(*
Nazwa:			FB_CapFeederV2
Opis:			Sorter nasadek i podajnik nasadek z podnośnikiem JIESANG
Wersja:			v0.1
Data:			2022-07-07
Autor:			DJA
Urzadzenia:		Silnik sortera, podnośnik JIESANG, Wydmuch, czujniki zapełnienia rękawa
Konfiguracja:	
Info:
-poprawiona wersja sortera względem poprzedniej, przerobione na aktualny standard State i RunningState
*)


FUNCTION_BLOCK FB_CapFeeder_old
VAR_INPUT
	
	bEnable						: BOOL;					//Zezowlenie na pracę stacji sprawdzania
	bEStop						: BOOL;					//Stop Awaryjny nieaktywny
	bRun						: BOOL;					//Włączenie sortera nasadek
	bHoming						: BOOL;					//Zezwolenie na wykonanie bazowania i pozycjonowania stacji sprawdzania
	bHeightSet					: BOOL;					// Bit do bazowania stacji na ustaloną wysokość 
	bIgnoreError				: BOOL;					//Ignorowania błędów cyklu pracy
	bReset						: BOOL;					//Reset błędu, jeśli w stanie "eError"
	lrHeightMotorPositionSV		: LREAL;				//Wysokość zadana na której ma znajdować się stacja
	lrMaxHeight					: LREAL;				//Maksymalna wysokość stacji sprawdzania
	lrMinHeight					: LREAL;				//Minimalna wysokość stacji sprawdzania
	bSorterCapSensor 			: BOOL;					// Wejście z czujnika ultradzwiękowego nasadki sortera
	bFullSleeveSensor			: BOOL;					// Wejście przepełnienia rękawa sortera
	bLevelSensor				: BOOL;					// Czujnik poziomu
	bHomingSensor				: BOOL;					// Wejscie czujnika bazowania napedu 
	iTimeDelayOn				: INT; 					//Czas na właczenie silnika sortera po zaniku sygnału przepełnienia z rękawa
	iTimeDelayOff				: INT; 					// Czas na wylączenie silnika sortera po wykryciu sygnału przepełnienia z rękawa sortera
	iTimeToEmptySleeveError		: INT;					// Czas do włączenia alrmu pustego rękawa
	bEngineOK					: BOOL;					//Wejście czujnika zabezpieczenia silnika 
	InEngineVelocityCV 			: UDINT;		
	InEngineSTW 				: UINT; 				// Statusword transportera wejściowo wyjściowego
	IbEngineWcState				: BOOL; 				// Statusword transportera wejściowo wyjściowego
	bHeightMotorEncoderPulse 	: BOOL;					//Sygnał impulsów enkodera siłownika
	rHeightMotorPositionOffset 	: REAL;					//Wysokość bazowania podnośnika
	bManualMovement				: BOOL; 				//Uruchomienie trybu ruchów ręcznych
	udiStationIndex				: UDINT;				// Indywidualny numer stacji
	sStationName				: STRING;				// Nazwa stacji
	
	tGatesFreq					:	TIME;
	
	bSensorInPipe				:	BOOL;				// Czujnik obecnośći flipflopa w rękawie
END_VAR

VAR_OUTPUT
	eState						: E_Station;			// Aktualny stan stacju
	eRunningState				: E_CapFeederState;		// Stan pracy stacji
	eRunningStateBeforeEstop	: E_CapFeederState;  	// Stan przed Estope
	bError						: BOOL;					// Błąd stacji
	udiErrorID					: UDINT;				// Nr blędu przeciągania formatek
	sErrorDescription			: STRING(200);			// Opis błędu
	sErrorDescription2			: STRING(200);			// Opis błędu
	sErrorStationName			: STRING;				// Nazwa stacj
	udiStationID				: UDINT;				// Nr stacji

	lrHeightMotorPositionCV		: LREAL;				//Aktualna pozycja podnośnika stacji
	bHeightMotorUp				: BOOL;					//Sterowanie silnikiem podnośnika  - RUCH W GÓRĘ
	bHeightMotorDown			: BOOL;					//Sterowanie silnikiem podnośnika  - RUCH W DÓŁ
	bSorterEngine 				: BOOL; 				// Sterowanie silnikiem sortera
	QnEngineVelocitySV 			: UDINT; 				// Nastawa prędkości
	QnEngineCTW 				: UINT;  				// Controlword transportera we/wy	
	bSorterAir 					: BOOL; 				// Sterowanie szybkim zaworem wydmuchu
	bHomingNeeded				: BOOL;					// Wymagane ponowne bazowanie (blad podczas bazowania lub stop awaryjny)
	bHomingDone					: BOOL;					// Stacja zbazowana 
	bCycleDone					: BOOL;					// Sygnał o zakończeniu cyklu
	bCycleNotDone				: BOOL;					// Sygnał o niezakończonym cyklu
	tCycleTime					: TIME;	 				// Czas cyklu 
	sWarningDescription			: STRING;
	bWarning1					: BOOL;
	udiWarningID				: UDINT;
	
	bGate1						:	BOOL;	//Szlaban w podajniku nakrętek #1
	bGate2						:	BOOL;	//Szlaban w podajniku nakrętek #2
	
END_VAR

VAR_IN_OUT
	bManualHeightMotorUp		: BOOL;					//Ruch ręczny podnośnika stacji w górę
	bManualHeightMotorDown		: BOOL;					//Ruch ręczny podnośnika stacji w dół
	bManualSorterEngine			: BOOL;					//Ręczne włączenie silnika sortera
	bManualSorterAir			: BOOL;					//Ręczne włączenie zaworu wydmuchu
	
	bManualGate1				:	BOOL;									// Szlaban #1 w rękawe
	bManualGate2				:	BOOL;									// Szlaban #2 w rękawe		
END_VAR

VAR
	i							:	INT;
	aBufferedSensorValue		:	ARRAY[0..50] OF BOOL;	
	iValvesCycleCase			:	INT;
	rtOutSensor					:	R_TRIG;

	// State
	eLastState					: E_Station;			//Stan ogólny bloku
	eLastStateTemp				: E_Station;			//Stan ogólny bloku
	eLastRunningState			: E_CapFeederState;		//Stan podbloku
	eLastRunningStateTemp		: E_CapFeederState;		//Stan podbloku

	fbHeightMotorEncoder		: FB_JiesangActuatorEncoder;				// Blok enkodera podnośnika chwytaka stabilizującego pod zakręcarką	
	bHeightMotorEncoderCounterReset						:BOOL; 				// Sygnał resetu enkodera
	lrLastHeightMotorPositionCV		: LREAL;				// Pozycja podnośnika w poprzednim cyklu programu
	bHeightMotorEncoderHomed	: BOOL;					// Informacja od enkodera że jest zbazowany		
	bStateError					: BOOL;
	
	tofHeightMotorDown			: TOF;					// Opóźnienie ruchu w dół, żeby nie przeciązać rozruchem układu
	rtEncoderHomed				: R_TRIG;				// Bit zakończenia enkodera
		
	tonHeightNoChange			: TON; 					// Timer wykrycia braku ruchu siłownika zmiany wysokości stacji
	tonHeightNoChangeTime		: TON; 					// Timer wykrycia braku ruchu siłownika zmiany wysokości stacji
	
	tonLimitPosMinReachedDelay	: TON;					// Timer osoiągniecia minimalnej wyskości 
	tonLimitPosMaxReachedDelay	: TON;					// Timer osiągnięcia maksymalnej wyskości
	tonSortingEngineOn			: TON;					// Opóźnienie po załączeniu napędu
	tonSortingEngineOff			: TON;					// Opóźnienie wyłączenia napędu
	tonSleeveFullEngineOn		: TON;					// Czas załączenia napędu po wykrciu braku nasadek
	tonEngineBlocked			: TON;					// Zablokowany silnik	
	rtCapSorterSensor			: R_TRIG;				// Triger
	tonTryUnblockWheel			: TON;					// Czas ruchu falownika w drugą stronę
	tofCapFeederSorterCapSensor	: TOF;					// Opóźnienie sygnału z czujnika obecności nasadki ultradzwiek
	tonCapFeederSorterCapSensor	: TON;					// Opóźnienie sygnału z czujnika obecności nasadki ultradźwięk
	tonAirBeforeStart			: TON;					// Czasówka opóźeniani przedmuchu
	tonAirBeforeStart2			: TON;					// Czasówka opóźeniani przedmuchu
	tonAirAfterStop				: TON;					// Czasówka przedmuchu po zatrzymaniu
	tonStoppingTime				: TON;					// Czasówka zbyt długiego zatrzymawania

	
	tonErrorHeightChange		: TON; 					// Timer błędu zacięcia się podnośnika
	tonEmptySleeveError			: TON;					// Timer pustego rękawa
	tonMaxHeightError			: TON;					// Timer ustawienia zbyt dużej wysokości stacji
	tonMinHeightError			: TON;					// Timer ustawienia zbyt małej wysokości stacji
	tonCycleTimer				: TON;					// Czasówka cyklu
	rtrigCycleTimerRead			: R_TRIG;				// Trigger do statystyk cyklu 
	
	tonSorterEngineError: TON;
	tonHomingSensor: TON;
	TimerOn: TON;
	TimerOff: TON;
	bImpOn: BOOL;
	rtCapFeederSorterCapSensor: R_TRIG;
	bBlowDelay: BOOL;
	tonbBlowDelay: TON;
	
	fbInverter: FB_MitsubishiInverter;
	tonInverterError: TON;
	(*Ostrzeżenia*)
	fbbLevelSensor:	FB_InputFilter;
	(*Inne*)	

	tonGates1	:	TON;	//Czasówka dla szlabanów w rękawe
	tonGates2	:	TON;	//Czasówka dla szlabanów w rękawe
	tonGates3	:	TON;	//Czasówka dla szlabanów w rękawe
	tonGates4	:	TON;	//Czasówka dla szlabanów w rękawe

		
	bGates	    :	BOOL;	//Controla szłabanow w rękawe  
	bTryUnblockWheel : BOOL;
	iTryUnblockWheel : INT;
END_VAR

//Wywołanie bloczków od stacji. Ważna jest ich kolejność!!!
ACT_Limits();
ACT_HeightMotor();
ACT_ErrorHandling();

ACT_Signals();
ACT_Control();
ACT_Inverter();
ACT_Statistic();
ACT_Status();
ACT_Warnings();
aStationID();	

lrLastHeightMotorPositionCV:=lrHeightMotorPositionCV;

ACTION ACT_Control:
	(*****Wyłączenie enable*****)
	IF NOT bEnable THEN
		IF eState <> E_Station.eDisabled AND eState <> E_Station.ePreparingToDisable THEN
				eState 				:= E_Station.ePreparingToDisable; 
		END_IF	
	END_IF

	(*****Estop*****)
	IF NOT bEstop  THEN	
		IF eState <> E_Station.eAborted AND eState <> E_Station.eAborting AND eState <> E_Station.eDisabled THEN
				eState 				:= E_Station.eAborting; 
		END_IF
	END_IF


	CASE eState OF
//--------------------------------------------------------------------------------
// Stan maszyny po wyłączeniu i przygotowanie do uruchomienia
	E_Station.eDisabled: 					// Stan nieaktywnosci (Stacja wyłączona) 
	
		IF bEnable THEN
			eState 				:= E_Station.ePreparingToReady; 
		END_IF 
		
//--------------------------------------------------------------------------------
// Stan maszyny po zatrzymaniu awaryjnym   
	E_Station.eAborted: 					// Stan bezpiecznego zatrzymania (po Abortingu) 

		IF bEStop THEN
			eState 				:= E_Station.ePreparingToReady;
		END_IF
		
//--------------------------------------------------------------------------------
// Stan maszyny naciśnieciu estopa 	
	E_Station.eAborting:                 	// Stan bezpiecznego zatrzymywania (po EStopie)
		bGate1:= FALSE;
		bGate2:= FALSE;
	
		ACT_ResetCommands();

		eState 						:=  E_Station.eAborted;  
		eRunningState				:=	E_CapFeederState.eReady;
		
//--------------------------------------------------------------------------------
// Stan masyzny po wykryciu błędu			
	E_Station.eError:                 	 	// Stan błędu 	
		
		ACT_ResetCommands();
		
		IF bReset THEN
			eState 				:= E_Station.eResetting;
			bError := FALSE;
		END_IF
		
//--------------------------------------------------------------------------------
// Stan masyzny po wykryciu błędu
	E_Station.eResetting:					// Stan resetowania bledu (po Errorze)
			CASE udiErrorID-udiStationIndex OF
		
				//Error 8 - Błąd falownika
				266:
					fbInverter.bReset	:= TRUE;
					bError 				:= FALSE;
				ELSE
					bError := FALSE;	
			END_CASE		
		
		IF NOT bError AND fbInverter.eState = E_Station.eReady THEN
			fbInverter.bReset	:= FALSE;	
			
			udiErrorID 			:=	0;
			sErrorDescription 	:=	'';
			eState 				:=	E_Station.ePreparingToReady;
			eRunningState		:=	E_CapFeederState.eReady;
		ELSE
			eState 				:=	E_Station.eError;
		END_IF
    
//--------------------------------------------------------------------------------
// Stan ruchoow manualnych
	E_Station.eManualMovement:     			// Stan ruchów manualnych  
   
		ACT_ManualMovements();
		//Wyjście z trybu serwisowego
		IF NOT bManualMovement THEN
			
			bHeightMotorUp				:=	FALSE;
			bHeightMotorDown			:=	FALSE;
			
			eState:=E_Station.eReady;
		END_IF
		

//--------------------------------------------------------------------------------
// Stan rozpoczecia bazowania
	E_Station.eHoming:						// Stan bazowania 
		
		ACT_Homing();
		IF NOT bHoming AND NOT bHeightSet THEN
			bHeightMotorDown					:=	FALSE;
			bHeightMotorUp						:=	FALSE;
		   eState								:=E_Station.ePreparingToReady;
		END_IF		
		
//--------------------------------------------------------------------------------
// Stan zakończenia bazowania
	E_Station.eHomingDone:                  // Stan wykonania bazowania 
	
		bHeightMotorDown					:=	FALSE;
		bHeightMotorUp						:=	FALSE;
		bHeightMotorEncoderCounterReset		:=	FALSE;
		bHomingDone							:=	TRUE;
		IF NOT bHoming AND NOT bHeightSet THEN
		   eState:=E_Station.eReady;
		END_IF
		
//--------------------------------------------------------------------------------
// Stan przygotowania do gotowości
	E_Station.ePreparingToReady:            // Stan przygotowywania do gotowosci (zawsze przed Ready)  
		
		bGate1:= FALSE;
		bGate2:= FALSE;
	
		bSorterEngine:=FALSE;
		bSorterAir:=FALSE;
		
		eRunningState:=E_CapFeederState.eReady;
		eState:=E_Station.eReady;	
		
//-------------------------------------------------------------------------------
// Stan przygotowania do wyłączenia maszyny
	E_Station.ePreparingToDisable:          // Stan przygotowywania do nieaktywnosci (po wyłączeniu Enable) 
		
		bGate1:= FALSE;
		bGate2:= FALSE;
	
		bSorterEngine:=FALSE;
		bSorterAir:=FALSE;
		bHeightMotorUp:= NOT tonHomingSensor.Q;
		bHeightMotorDown:=FALSE;	
		IF tonHeightNoChange.Q OR tonHeightNoChangeTime.Q THEN
			bHeightMotorUp			:=	FALSE;
			bHeightMotorDown		:=	FALSE;	
			eRunningState			:=	E_CapFeederState.eReady;		
			eState					:=	E_Station.eDisabled;
		END_IF	
			
//--------------------------------------------------------------------------------
// Stan gotowości
	E_Station.eReady:						// Stan gotowosci 
	
		IF bRun AND NOT bCycleDone AND NOT bCycleNotDone THEN
			eState 				:= E_Station.eStarting; 
		END_IF
		IF bHoming OR bHeightSet THEN
			bHomingDone							:=	FALSE;
			eState 								:= E_Station.eHoming; 
		END_IF
		IF bManualMovement THEN
			//Jeśli przejście w tryb ruchów manualnych przepisz wszystkie stany siłowników sterowanych przez moduł
			//aby zapobiec ewentualnym kolizjom po wejściu w tryb serwisowy
			
			bManualHeightMotorUp		:= bHeightMotorUp;
			bManualHeightMotorDown		:= bHeightMotorDown;
			
			eState 						:= E_Station.eManualMovement; 
		END_IF
		IF NOT bRun THEN
			bCycleDone 			:= FALSE;
			bCycleNotDone 		:= FALSE;			
		END_IF
		
//--------------------------------------------------------------------------------
// Stan zatrzymywania
	E_Station.eStopping:					// Stan zatrzymywania 
		
		bSorterAir 		:= 	TRUE;
		bSorterEngine 	:=	FALSE;
		IF tonStoppingTime.Q THEN
			ACT_ResetCommands();
			eRunningState							:= E_CapFeederState.eReady;
			eState									:= E_Station.eReady;
		END_IF

		
//--------------------------------------------------------------------------------
// Stan uruchomienia lini ( po eReady)
	E_Station.eStarting:                  	// Stan uruchamiania (po Ready)
		iValvesCycleCase		:=0;
		eState					 := E_Station.eRunning; 

//--------------------------------------------------------------------------------
// Stan wykonywania pracy
	E_Station.eRunning:               		// Stan wykonywania cyklu (po Startingu), w tym stanie osobny

		ACT_Running();
		IF NOT bRun THEN 					(*Przerywanie cyklu*)
			eState				:= E_Station.eStopping;
			//bCycleNotDone		:= TRUE;
		END_IF
		(*IF bCycleDone OR bCycleNotDone THEN (*Cykl zakończony*)
			eState 				 := E_Station.eReady;
		END_IF*)						
		
		
END_CASE
END_ACTION

ACTION ACT_ErrorHandling:
//OBSŁUGA BŁĘDÓW STACJI SPRAWDZANIA
//************LISTA BŁĘDÓW***************
bStateError:= (eState=E_Station.eError) OR (eState=E_Station.eResetting) OR bIgnoreError;

//************LISTA BŁĘDÓW***************

//Error 1 - podnośnik nie porusza się pomimo wysterowania 
tonErrorHeightChange(IN:=(bHeightMotorUp OR bHeightMotorDown) AND lrLastHeightMotorPositionCV=lrHeightMotorPositionCV, PT:=T#3S);
tonEmptySleeveError(IN:=NOT bFullSleeveSensor AND bRun, PT:=INT_TO_TIME(iTimeToEmptySleeveError)*1000); //Było 30, teraz jest z receptur
tonMaxHeightError(IN:=lrHeightMotorPositionSV>lrMaxHeight AND NOT bHomingNeeded AND eState=E_Station.eReady,PT:=T#30S);
tonMinHeightError(IN:=lrHeightMotorPositionSV<lrMinHeight AND NOT bHomingNeeded AND eState=E_Station.eReady,PT:=T#30S);
tonSorterEngineError(IN:= NOT bEngineOK AND bSorterEngine, PT:=T#3S);
tonInverterError(IN:=fbInverter.bError AND NOT bStateError, PT:=T#3S);

IF (bEnable OR (eState = E_Station.ePreparingToDisable)) AND NOT bIgnoreError THEN
	
	IF tonErrorHeightChange.Q THEN
		bError:=TRUE;
		udiErrorID:=261;
		//udiErrorID:= udiErrorID+udiStationIndex;
		sErrorDescription:='Blokada podnośnika lub brak zasilania - sprawdź czujnik lub odblokuj mechanicznie';	
		sErrorDescription2:='';
	END_IF
	
	
	IF tonSorterEngineError.Q THEN
		bError:=TRUE;
		udiErrorID:=262;
		//udiErrorID:= udiErrorID+udiStationIndex;
		sErrorDescription:='Bład zabezpieczenia silnika - sprawdź wyłącznik';	
		sErrorDescription2:='';	
	END_IF
	
	//Error 3 - Pusty rekaw sortera nasadek
	IF tonEmptySleeveError.Q THEN
		bError:=TRUE;
		udiErrorID:=263;
		//udiErrorID:= udiErrorID+udiStationIndex;
		sErrorDescription:='Pusty rękaw sortera - uzupełnij nasadki';
		sErrorDescription2:='';
	END_IF
	
	
	//Error 4 - Bład nastaw max
	IF tonMaxHeightError.Q  THEN
		bError:=TRUE;
		udiErrorID:=264;
		//udiErrorID:= udiErrorID+udiStationIndex;
		sErrorDescription:='Wartość zadana wysokości jest większa od maksymalnej - zmień ustawienia w recepturze';
		sErrorDescription2:=REAL_TO_STRING(LREAL_TO_INT(lrMaxHeight));
	END_IF
	
	//Error 5 - Bład nastaw min
	IF tonMinHeightError.Q THEN
		bError:=TRUE;
		udiErrorID:=265;
		//udiErrorID:= udiErrorID+udiStationIndex;
		sErrorDescription:='Wartość zadana wysokości jest mniejsza od minimalnej - zmień ustawienia w recepturze ';
		sErrorDescription2:=REAL_TO_STRING(LREAL_TO_INT(lrMinHeight));
	END_IF	
	
	//Error 6 - Bład falownika
	IF tonInverterError.Q THEN
		bError:=TRUE;
		udiErrorID:=266;
		//udiErrorID:= udiErrorID+udiStationIndex;
		sErrorDescription:='Błąd falownika';
		sErrorDescription2:='';
	END_IF		
	
	
	
ELSE
	bError	:=FALSE;
END_IF


//-----------------------------------------------------------------------
IF bError AND NOT bStateError THEN

	IF eLastState = eRunning THEN
		bCycleNotDone						:= TRUE;
	END_IF

	eState 									:= E_Station.eError;
END_IF


//------------------------------------------------------------------------

(*Wyświetlanie błedu na wyjściu*)
bError;

(*Przepisywanie nazwy stacji*)
sErrorStationName 							:= sStationName;

//Jezeli nie zbazowane to potrzebne bazowanie
IF NOT bHeightMotorEncoderHomed  THEN
	bHomingDone								:=	FALSE;
END_IF
END_ACTION

ACTION ACT_HeightMotor:
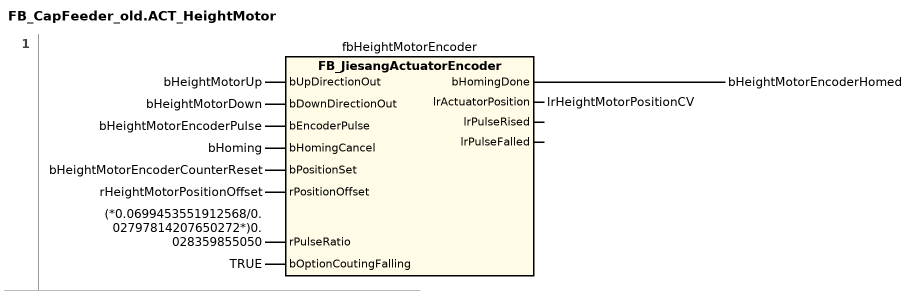
// NETWORK 1
fbHeightMotorEncoder(
    bUpDirectionOut := bHeightMotorUp,
    bDownDirectionOut := bHeightMotorDown,
    bEncoderPulse := bHeightMotorEncoderPulse,
    bHomingCancel := bHoming,
    bPositionSet := bHeightMotorEncoderCounterReset,
    rPositionOffset := rHeightMotorPositionOffset,
    rPulseRatio := (*0.0699453551912568/0.02797814207650272*)0.028359855050,
    bOptionCoutingFalling := TRUE,
    lrActuatorPosition => lrHeightMotorPositionCV); // FB_JiesangActuatorEncoder
bHeightMotorEncoderHomed := fbHeightMotorEncoder.bHomingDone;
END_ACTION

ACTION ACT_Homing:
//BAZOWANIE

tofHeightMotorDown(IN:=bHeightMotorDown, PT:=T#1S); //Zabezpieczenie przed zbyt szybkim przełączeniem pomiędzy Down a Up, bezpiecznieki sie palą
	
//Podnoszenie stacji do maksymalnej pozycji
IF NOT bHeightMotorEncoderHomed OR rtEncoderHomed.Q THEN
	bHeightMotorUp:=(*TRUE*) NOT tofHeightMotorDown.Q AND NOT tonHomingSensor.Q;
	bHeightMotorDown:=FALSE;
	IF tonHeightNoChange.Q OR tonHeightNoChangeTime.Q THEN
		bHeightMotorEncoderCounterReset:=TRUE;
		bHeightMotorUp:=FALSE;
    END_IF
	//Jesli enkoder zbazowany zakończ bazowanie	
	IF rtEncoderHomed.Q  THEN
		bHeightMotorUp:=FALSE;
		bHeightMotorDown:=FALSE;
		eState:=E_Station.eHomingDone;
	END_IF		
		
//Po podniesieniu stacji opuszczanie do ustalonej wysokości
ELSIF bHeightMotorEncoderHomed THEN
	bHeightMotorEncoderCounterReset:=FALSE;
	bHeightMotorUp:=lrHeightMotorPositionCV<=lrHeightMotorPositionSV;
	bHeightMotorDown:=lrHeightMotorPositionCV>=lrHeightMotorPositionSV;
	//Kiedy stacja osiągnie wysokość zadaną
	IF ABS(lrHeightMotorPositionCV-lrHeightMotorPositionSV)<0.5 OR tonLimitPosMaxReachedDelay.Q OR tonLimitPosMinReachedDelay.Q THEN
		bHeightMotorDown:=FALSE;
		bHeightMotorUp:=FALSE;
		eState:=E_Station.eHomingDone;
	END_IF			
END_IF
END_ACTION

ACTION ACT_Inverter:
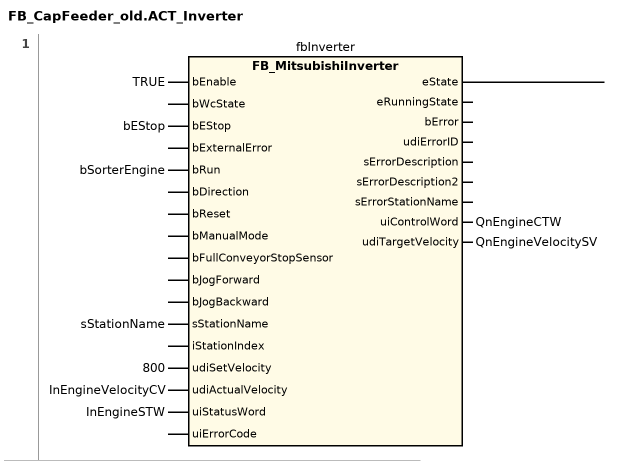
// NETWORK 1
fbInverter(
    bEnable := TRUE,
    bEStop := bEStop,
    bRun := bSorterEngine,
    sStationName := sStationName,
    udiSetVelocity := 800,
    udiActualVelocity := InEngineVelocityCV,
    uiStatusWord := InEngineSTW,
    uiControlWord => QnEngineCTW,
    udiTargetVelocity => QnEngineVelocitySV); // FB_MitsubishiInverter
END_ACTION

ACTION ACT_Limits:
IF iTimeToEmptySleeveError < 5 THEN
	iTimeToEmptySleeveError := 5;
END_IF
END_ACTION

ACTION ACT_ManualMovements:
//W trybie ruchów manualnych wykonuj ruchy za pomocą rozkazów manualnych
IF NOT bRun THEN
	
	bHeightMotorUp:=bManualHeightMotorUp;
	bHeightMotorDown:=bManualHeightMotorDown;
	bSorterEngine:=bManualSorterEngine;
	bSorterAir:=bManualSorterAir;
	
	bGate1:=bManualGate1; //Not dla tego, że defoltowy stan WYSUNIĘTY (true)
	bGate2:=bManualGate2; //Not dla tego, że defoltowy stan WYSUNIĘTY (true)

(*ELSE	//Kasuje zeby po cyklu nic sie nie poruszało

	bManualHeightMotorUp 	:= FALSE;
	bManualHeightMotorDown  := FALSE;
	bSorterEngine	:=FALSE;
	bSorterAir		:=FALSE;
*)	
END_IF


IF bHoming OR bHeightSet THEN
	eState:=E_Station.eHoming;
END_IF

IF bRun THEN	
	ACT_Running();
END_IF
//Zabezpieczenie przed kolizją stacji poprzez ruch podnośnika	
IF bHeightMotorDown AND lrHeightMotorPositionCV<=lrMinHeight AND NOT bHoming AND NOT bHeightSet THEN
	bHeightMotorDown:=FALSE;
END_IF	

IF bHeightMotorUp AND lrHeightMotorPositionCV>=lrMaxHeight AND NOT bHoming AND NOT bHeightSet THEN
	bHeightMotorUp:=FALSE;
END_IF
END_ACTION

ACTION ACT_ResetCommands:
//Reset komend ruchu 	


bHeightMotorUp				:=	FALSE;
bHeightMotorDown			:=	FALSE;
bSorterAir 		:= 	FALSE;
bSorterEngine 		:=	FALSE;
END_ACTION

ACTION ACT_Running:
//----------------------------------------------------------------------------------
// Obsługa podajnik zamknięc


(*CASE iValvesCycleCase OF
	0:
		bGate1:= FALSE;
		IF (tonGates1.Q) THEN
			iValvesCycleCase :=1;
		END_IF
	1:
		bGate1:= TRUE;
		IF (tonGates2.Q) THEN
			iValvesCycleCase :=2;
		END_IF	
	2:
		bGate2:= FALSE;
		IF (tonGates3.Q) THEN
			iValvesCycleCase :=3;
		END_IF
	3:
		bGate2:= TRUE;
		IF (tonGates4.Q) THEN
			iValvesCycleCase :=0;
		END_IF	
END_CASE*)

//rtOutSensor(CLK:=P08_CapSorter.IbCapSorterGateGateAfterSensor);
	
CASE iValvesCycleCase OF
	0:
		//IF (rtOutSensor.Q) THEN
		IF (NOT bSensorInPipe) THEN

			iValvesCycleCase:=1;
		END_IF
		;
	1:
		bGate1:= TRUE;
		IF (tonGates1.Q) THEN
			iValvesCycleCase :=2;
		END_IF
	2:
		bGate1:= FALSE;
		IF (tonGates2.Q) THEN
			iValvesCycleCase :=3;
		END_IF	
	3:
		bGate2:= TRUE;
		IF (tonGates3.Q) THEN
			iValvesCycleCase :=4;
		END_IF
	4:
		bGate2:= FALSE;
		IF (tonGates4.Q) THEN
			iValvesCycleCase :=0;
		END_IF	
END_CASE

CASE eRunningState OF
	
	//NIEGOTOWY
	E_CapFeederState.eDisabled:
		eRunningState:=E_CapFeederState.eReady;

	E_CapFeederState.eReady:
		iTryUnblockWheel		:=	0;
		bTryUnblockWheel		:= FALSE;	
		fbInverter.bDirection 	:= FALSE;
		IF bRun THEN
			eRunningState			:=E_CapFeederState.eSorting;
		END_IF
	
	
	E_CapFeederState.eSorting:
	
		bSorterEngine:=tonAirBeforeStart.Q;
		bSorterAir:=(	//Nie wiem co to za wymysły
						(aBufferedSensorValue[20](*tofCapFeederSorterCapSensor.Q*) OR NOT tonAirBeforeStart2.Q)(* AND bImpON*)AND NOT bBlowDelay
					)	OR	
					bTryUnblockWheel // Dmuchanie jeżeli jest obrót do tyłu
;
		//aBufferedSensorValue[20] - 20 to jest opóznenie (buferizacja signala czujnika w cyklach programy (3ms x 20 = 60 ms). Czas opóznenia 
		//możemy obliczyć od prędcosci falownika i prszykładni: mamy 51 gniazdk0, 800 rpm, przykladnia 1:40 => mamy 800/40=20rmp, /60 =>
		//0,33 obrota / sec => 0,33 obrota/sec * 51 dnazdko/obrot = 17 gniazdek/sek => 1/17 = 0,059sec/1gniazdko => opoznenie 60 ms
		//60ms/3ms(czas cyclu) => 20 cyclów
		
		(*Próba odblokowania koła*)
			iTryUnblockWheel := iTryUnblockWheel + 1;
			IF rtCapSorterSensor.Q THEN
				iTryUnblockWheel	:=	0;
			END_IF
			IF tonEngineBlocked.Q THEN
				bTryUnblockWheel := TRUE;
			END_IF	
			IF bTryUnblockWheel THEN
				fbInverter.bDirection := TRUE;
			END_IF
			IF tonTryUnblockWheel.Q THEN
				iTryUnblockWheel		:=	0;//dp
				bTryUnblockWheel		:= FALSE;
				fbInverter.bDirection 	:= FALSE;
			END_IF
		(* Koniec Próba odblokowania koła*)	
		
		IF tonSortingEngineOff.Q THEN 
			eRunningState 			:=E_CapFeederState.eSleeveFull;
		END_IF
	
	E_CapFeederState.eSleeveFull:
	
		bSorterEngine:=FALSE;
		bSorterAir:=NOT tonAirAfterStop.Q(* AND bImpON*);
		IF tonAirAfterStop.Q THEN
			IF tonSortingEngineOn.Q THEN
				eRunningState		:=E_CapFeederState.eSorting; 
			END_IF
		END_IF
	
	E_CapFeederState.eSleeveLowLevel:
	
			//Wlaczenie silnika i zaworu po czasie
		bSorterEngine:=TRUE;
		bSorterAir:=tofCapFeederSorterCapSensor.Q (*AND bImpON*);
		IF tonSortingEngineOff.Q THEN
			eRunningState		 	:=E_CapFeederState.eSorting;
		END_IF
	
END_CASE
END_ACTION

ACTION ACT_Signals:
(** Timery na potrzeby bazowania**)
rtEncoderHomed(CLK:=bHeightMotorEncoderHomed,Q=>);
tonHeightNoChange(IN:=((bHeightMotorUp OR bHeightMotorDown OR tonHomingSensor.Q) AND (lrLastHeightMotorPositionCV=lrHeightMotorPositionCV)), PT:=T#500MS); 
tonHomingSensor(IN:=(bHomingSensor), PT:=T#100MS);
//tonHeightNoChangeTime(IN:=(eState = E_Station.eHoming OR eState = E_Station.ePreparingToDisable) AND bHeightMotorUp, PT:=T#8S); 

tonLimitPosMinReachedDelay(IN:=(lrHeightMotorPositionCV<=lrMinHeight) AND eState=E_Station.eHoming,PT:=T#2S);
tonLimitPosMaxReachedDelay(IN:=(lrHeightMotorPositionCV>=lrMaxHeight) AND eState=E_Station.eHoming,PT:=T#2S);
	
(** Timery używane podczas pracy stacji**)
tonSortingEngineOff(IN:=((eRunningState=E_CapFeederState.eSorting OR eRunningState=E_CapFeederState.eSleeveLowLevel) AND bRun AND bFullSleeveSensor),PT:=INT_TO_TIME(iTimeDelayOff));
tonSortingEngineOn(IN:=((eRunningState=E_CapFeederState.eSorting OR eRunningState=E_CapFeederState.eSleeveFull) AND bRun AND NOT bFullSleeveSensor),PT:=INT_TO_TIME(iTimeDelayOn));
tonSleeveFullEngineOn(IN:=(eRunningState=E_CapFeederState.eSleeveFull AND bRun AND NOT bFullSleeveSensor),PT:=INT_TO_TIME(iTimeDelayOff));
rtCapSorterSensor(CLK:=bSorterCapSensor, Q=>);
tonEngineBlocked(IN:=iTryUnblockWheel > 1500 AND bSorterEngine AND NOT bTryUnblockWheel,PT:=T#1MS); //Zablokowany silnik
tonTryUnblockWheel(IN:=bTryUnblockWheel, PT:=T#1S900MS);
tofCapFeederSorterCapSensor(IN:=tonCapFeederSorterCapSensor.Q,PT:=T#10MS); //bylo 200
tonCapFeederSorterCapSensor(IN:=bSorterCapSensor,PT:=T#3mS);//było 3ms
tonAirBeforeStart(IN:=eRunningState=E_CapFeederState.eSorting, PT:=T#1S);
rtCapFeederSorterCapSensor(CLK:=tofCapFeederSorterCapSensor.Q,Q=>);

tonAirBeforeStart2(IN:=eRunningState=E_CapFeederState.eSorting, PT:=T#2S);
tonAirAfterStop(IN:=eRunningState=E_CapFeederState.eSleeveFull, PT:=T#2S);

//prszesunęcie wartosci czujnika po buforu opoznenia 

FOR i:=40 TO 1 BY -1 DO
	aBufferedSensorValue[i] := aBufferedSensorValue[i-1];
END_FOR
aBufferedSensorValue[0] := bSorterCapSensor;

IF rtCapFeederSorterCapSensor.Q THEN
	bBlowDelay := TRUE;
	
END_IF
tonbBlowDelay(IN:=bBlowDelay,PT:=T#35MS);
IF tonbBlowDelay.Q THEN
	bBlowDelay:= FALSE;
END_IF
TimerOn (IN := NOT bImpOn, PT := T#10MS);
IF TimerOn.Q THEN
	bImpOn := TRUE;
END_IF
TimerOff (IN := bImpOn, PT := T#10MS);
IF TimerOff.Q THEN
	bImpON := FALSE;
END_IF

//Czasówki pneumatiki
//tonGates1(IN:= (iValvesCycleCase = 0 AND (eState = E_Station.eRunning OR eState = E_Station.eManualMovement)), PT:=T#300MS);//150//300
//tonGates2(IN:= (iValvesCycleCase = 1 AND (eState = E_Station.eRunning OR eState = E_Station.eManualMovement)), PT:=T#200MS);//500//300
//tonGates3(IN:= (iValvesCycleCase = 2 AND (eState = E_Station.eRunning OR eState = E_Station.eManualMovement)), PT:=T#300MS);//150//300
//tonGates4(IN:= (iValvesCycleCase = 3 AND (eState = E_Station.eRunning OR eState = E_Station.eManualMovement)), PT:=T#200MS);//500//300

//Czasówki pneumatiki
tonGates1(IN:= (iValvesCycleCase = 1 AND (eState = E_Station.eRunning OR eState = E_Station.eManualMovement)), PT:=T#200MS);//150//300
tonGates2(IN:= (iValvesCycleCase = 2 AND (eState = E_Station.eRunning OR eState = E_Station.eManualMovement)), PT:=T#200MS);//500//300
tonGates3(IN:= (iValvesCycleCase = 3 AND (eState = E_Station.eRunning OR eState = E_Station.eManualMovement)), PT:=T#200MS);//150//300
tonGates4(IN:= (iValvesCycleCase = 4 AND (eState = E_Station.eRunning OR eState = E_Station.eManualMovement)), PT:=T#200MS);//500//300


(** Dodatkowy timer przy zatrzymywaniu**)
tonStoppingTime( IN:= eState= E_Station.eStopping, PT:=T#2S);
END_ACTION

ACTION ACT_Statistic:
//Statystyka do zliczania czasu cyklu 
rtrigCycleTimerRead(CLK:=eRunningState=E_CapFeederState.eSleeveFull OR eRunningState=E_CapFeederState.eSleeveLowLevel);

	IF rtrigCycleTimerRead.Q THEN
		tCycleTime:=tonCycleTimer.ET;
		
	END_IF
	
tonCycleTimer(IN:=eRunningState= E_CapFeederState.eSorting , PT:=T#1D);
END_ACTION

ACTION ACT_Status:

(*Zapisywanie ostatniego stanu*)
	IF eLastStateTemp<>eState THEN
		eLastState := eLastStateTemp;
	END_IF
	eLastStateTemp := eState;
	
	IF eLastRunningStateTemp<>eRunningState THEN
		eLastRunningState := eLastRunningStateTemp;
	END_IF
	eLastRunningStateTemp := eRunningState;
(*Koniec Zapisywanie ostatniego stanu*)
END_ACTION

ACTION ACT_Warnings:
//Usrawianie warningów

//Filtrowanie czujnika ultradźwiękowego
fbbLevelSensor	(bIN:=NOT bLevelSensor AND (eRunningState=E_CapFeederState.eSorting OR eRunningState=E_CapFeederState.eSleeveLowLevel OR eRunningState=E_CapFeederState.eSleeveFull) , tFilterTimeOn:= T#5S, tFilterTimeOff:=T#5S , bOUT=> );


IF fbbLevelSensor.bOUT THEN
		bWarning1						:=	TRUE;			
		udiWarningID					:=	1;
		sWarningDescription				:=	'Nieski poziom w sorterze nasadek';
ELSE
		bWarning1						:=	FALSE;			
		udiWarningID					:=	0;
		sWarningDescription				:=	'';
END_IF
END_ACTION

ACTION aStationID:
udiStationID	:=	udiStationIndex;
END_ACTION

END_FUNCTION_BLOCK

(* stored: Version 1.1.0.1, ProductVersion 3.1.4026.13, FileIdentifier 240dc6da26103993ab5526b7155bc7be91adafcf, FileSignature 1ca4b745385e66019a224ece77e967c43c3fe84dba80b17898fde0724878a7a76997b30f08615ec5983beb15829a89977eb7daa3440a2eca313e119eea2be2b3593b5629cd5f31ed2dcd6598bd82435a096fa9e286fdc61555022b88f3a5aa1df890d281bf979f109d001595518352a1fb0068e433110b9b500459019382e123236f3ae6da92a81d493fb07e4d71ad90379a0c4bc823404436f6ed4e690a5245ad54bfc1ddb94d5b3c8754dd36ae5c32a2f54fc818874f82480221fe7faa9eeef6676ca47a5be9f1ddea32431be39df2ae8ffcd6df16bddfe90df7846b59971957de5bf8ecd67249fcd2c1d249700d8b4ada32b58d7ecbfc6522c81fb07e36ba
   POU FB_CapFeeder_old: Id {c10c434b-7374-488b-aa42-9e04baf30261}, SpecialFunc None
   Action ACT_Control: Id {c2fc4ed5-e164-40a6-95f8-121e42585578}
   Action ACT_ErrorHandling: Id {94fcb7c9-af20-4929-a668-b8adf2341033}
   Action ACT_HeightMotor: Id {6db5a767-ab11-41f6-b596-e6b6dea62fd5}
   Action ACT_Homing: Id {f1494c96-6e62-419d-816d-7a92211eff67}
   Action ACT_Inverter: Id {a21b2afd-c7b7-497f-9e25-0e854e9a927d}
   Action ACT_Limits: Id {bb4aef5a-ef70-48dd-b217-23ac5f8ae19e}
   Action ACT_ManualMovements: Id {28244a7d-4e2d-4673-a342-ad49753b5afc}
   Action ACT_ResetCommands: Id {b323b2df-29d1-4847-964c-d64ea51b2727}
   Action ACT_Running: Id {6dcb117e-23b2-4547-bb97-27d285dbed74}
   Action ACT_Signals: Id {04190e77-0ee6-4f8d-b1ff-268791e3f63b}
   Action ACT_Statistic: Id {a11750b5-8b9c-45e7-a68c-888caa58fe35}
   Action ACT_Status: Id {6540c7f6-6515-4c98-9603-2a9f280a01a2}
   Action ACT_Warnings: Id {d6dea6f4-29b6-48ed-96b7-b75da90111d4}
   Action aStationID: Id {0f18d03e-6a87-4e44-892b-265e9df5954d} *)
